FUNCTION_BLOCK Ticksource
  (* Standard: 61499-2 *)
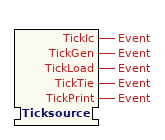
  EVENT_OUTPUT
    TickIc;
    TickGen;
    TickLoad;
    TickTie;
    TickPrint;
  END_EVENT
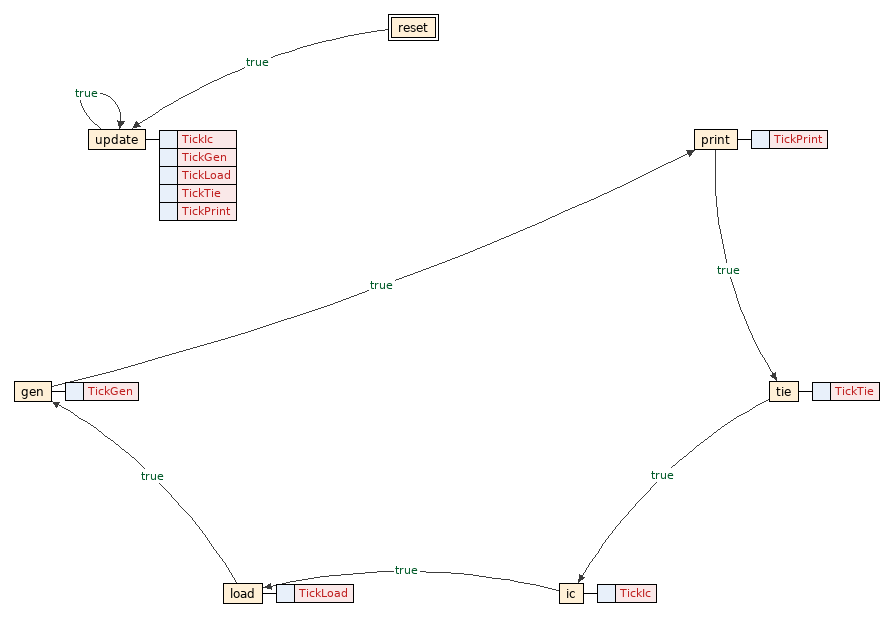
  EC_STATES
    reset;
    print : -> TickPrint;
    tie : -> TickTie;
    ic : -> TickIc;
    load : -> TickLoad;
    gen : -> TickGen;
    update : -> TickIc, -> TickGen, -> TickLoad, -> TickTie, -> TickPrint;
  END_STATES
  EC_TRANSITIONS
    reset TO update := true;
    print TO tie := true;
    tie TO ic := true;
    ic TO load := true;
    load TO gen := true;
    gen TO print := true;
    update TO update := true;
  END_TRANSITIONS
END_FUNCTION_BLOCK
